{attribute 'Tc2GvlVarNames'}
VAR_CONFIG
END_VAR

(* stored: Version 1.1.0.1, ProductVersion 3.1.0.26
   GVL Variable_Configuration: Id {4a7cda2d-82d1-4d35-9fa6-c02714fe2489} *)
